Fanuc KAREL source: FanucMonitorService.kl

PROGRAM FANUC_MONITOR_SERVICE
%NOLOCKGROUP
%NOPAUSE = ERROR + COMMAND + TPENABLE
%NOABORT = ERROR + COMMAND
%COMMENT = 'FANUC monitor TCP server'
%ENVIRONMENT sysdef
%ENVIRONMENT fdev
%ENVIRONMENT flbt
%ENVIRONMENT MOTN
%ENVIRONMENT REGOPE
%ENVIRONMENT TIM

VAR
  channel    : FILE
  status     : INTEGER
  entry      : INTEGER
  session_on : BOOLEAN
  seq        : INTEGER
  robot_ms   : INTEGER
  frame_ms   : INTEGER
  last_us    : INTEGER
  current_us : INTEGER
  delta_us   : INTEGER
  remain_us  : INTEGER
  done       : INTEGER
  pos        : XYZWPREXT
  jpos       : JOINTPOS
  vals       : ARRAY[9] OF REAL
  service_on : BOOLEAN
  stop_is_real : BOOLEAN
  stop_value : INTEGER
  stop_real : REAL
  done_is_real : BOOLEAN
  done_int     : INTEGER
  done_real    : REAL
  utool:POSITION
  uframe:POSITION
  out_pos:POSITION
  wjnt_cfg:CONFIG
  ext_ang:ARRAY[3] OF REAL
  pos_1:XYZWPR
  config_ref:INTEGER
  reg_status:INTEGER
  kine_status:INTEGER

ROUTINE InitMonitorPort
BEGIN
  SET_VAR(entry, '*SYSTEM*', '$HOSTS_CFG[5].$SERVER_PORT', 9001, status)
END InitMonitorPort

ROUTINE ClearStopFlag
BEGIN
  SET_INT_REG(99, 0, status)
END ClearStopFlag

ROUTINE CheckStopFlag
BEGIN
  GET_REG(99, stop_is_real, stop_value, stop_real, status)
  IF status = 0 THEN
    IF NOT stop_is_real THEN
      IF stop_value <> 0 THEN
        service_on = FALSE
        session_on = FALSE
      ENDIF
    ENDIF
  ENDIF
END CheckStopFlag

ROUTINE UpdateFrameTime
BEGIN
  current_us = GET_USEC_TIM
  delta_us = GET_USEC_SUB(current_us, last_us)
  IF delta_us < 0 THEN
    delta_us = 0
  ENDIF
  delta_us = delta_us + remain_us
  robot_ms = robot_ms + (delta_us DIV 1000)
  remain_us = delta_us MOD 1000
  last_us = current_us
  frame_ms = robot_ms
END UpdateFrameTime

ROUTINE UpdateDoneState
BEGIN
  done = -1
  GET_REG(98, done_is_real, done_int, done_real, status)
  IF status = 0 THEN
    IF done_is_real THEN
      done = -1
    ELSE
      IF done_int = 0 THEN
        done = 0
      ELSE
        done = 1
      ENDIF
    ENDIF
  ENDIF
END UpdateDoneState

ROUTINE WriteMonitorFrame(ch : FILE)
BEGIN
  vals[1] = 0.0
  vals[2] = 0.0
  vals[3] = 0.0
  vals[4] = 0.0
  vals[5] = 0.0
  vals[6] = 0.0
  vals[7] = 0.0
  vals[8] = 0.0
  vals[9] = 0.0

  UpdateDoneState
  UpdateFrameTime
  pos_1 = CURPOS(0, 0)
  jpos = CURJPOS(0, 0)
  reg_status = 0
  utool = GET_POS_REG(3, reg_status) -- 获得PR[3]的工具坐标
  IF reg_status = 0 THEN
    uframe = GET_POS_REG(4, reg_status) -- 获得PR[4]的用户坐标
  ENDIF
  CNV_JPOS_REL(jpos, vals, status)
  config_ref = 0
  IF reg_status = 0 THEN
    JOINT2POS(jpos, uframe, utool, config_ref, out_pos, wjnt_cfg, ext_ang, kine_status)
    IF kine_status = 0 THEN
      pos = out_pos
    ELSE
      pos = pos_1
    ENDIF
  ELSE
    pos = pos_1
  ENDIF

  WRITE ch('MON:',
           seq, ',',
           frame_ms, ',',
           done, ',',
           pos.x::10::3, ',',
           pos.y::10::3, ',',
           pos.z::10::3, ',',
           pos.w::10::3, ',',
           pos.p::10::3, ',',
           pos.r::10::3, ',',
           vals[1]::10::3, ',',
           vals[2]::10::3, ',',
           vals[3]::10::3, ',',
           vals[4]::10::3, ',',
           vals[5]::10::3, ',',
           vals[6]::10::3, ',',
           vals[7]::10::3, ',',
           vals[8]::10::3, ',',
           vals[9]::10::3, CR)
END WriteMonitorFrame

BEGIN
  service_on = TRUE
  seq = 0
  robot_ms = 0
  frame_ms = 0
  remain_us = 0
  last_us = GET_USEC_TIM
  SET_FILE_ATR(channel, ATR_IA)
  InitMonitorPort
  ClearStopFlag
  WRITE('FANUC monitor TCP server started', CR)
  WRITE('Mode: ROBOT=SERVER, PC=CLIENT, TAG=S5:, PORT=9001', CR)

  WHILE service_on DO
    MSG_CONNECT('S5:', status)
    WRITE('MON MSG_CONNECT STATUS=', status, CR)
    IF status <> 0 THEN
      CheckStopFlag
      DELAY(500)
    ELSE
      WRITE('Waiting for TCP client on S5 port 9001...', CR)
      CLR_IO_STAT(channel)
      OPEN FILE channel('rw', 'S5:')
      status = IO_STATUS(channel)
      IF status = 0 THEN
        WRITE('Monitor client connected', CR)
        last_us = GET_USEC_TIM
        remain_us = 0
        session_on = TRUE
        WHILE session_on DO
          WriteMonitorFrame(channel)
          status = IO_STATUS(channel)
          IF status <> 0 THEN
            session_on = FALSE
          ELSE
            seq = seq + 1
            CheckStopFlag
            DELAY(50)
          ENDIF
        ENDWHILE
        CLOSE FILE channel
        CLR_IO_STAT(channel)
        WRITE('Monitor client disconnected', CR)
      ELSE
        WRITE('OPEN S5 STATUS=', status, CR)
        CLR_IO_STAT(channel)
      ENDIF
      CLR_IO_STAT(channel)
      MSG_DISCO('S5:', status)
      WRITE('MON MSG_DISCO S5 STATUS=', status, CR)
      DELAY(500)
    ENDIF
  ENDWHILE

  MSG_DISCO('S5:', status)
  WRITE('FANUC monitor TCP server stopped', CR)
END FANUC_MONITOR_SERVICE
